(* Schneider Machine Expert - Basic project 13_counter_simulation, file version 3.0.0.0 *)
(* ProjectInformations: Name=New project *)

HARDWARE
  Cpu 0: TM221CE16R
  EthernetConfiguration: NetworkName=M221, IpAllocationMode=FixedAddress, IpAddress=0.0.0.0, SubnetMask=0.0.0.0
  SerialLineConfiguration: Baud=Baud19200, Parity=ParityEven, DataBits=DataBits8, StopBits=StopBits1, PhysicalMedium=PhysicalMediumRs485, TransmissionMode=TransmissionModeModbusRtu, SlaveId=1, Addressing=SlaveAddressing
  MastTask: UsePeriodScanMode=false, PeriodScan=100
  FastTask: Period=255
  CpuBehavior: StartingMode=StartAsPreviousState, AutoSaveRamOnEeprom=true, WatchdogPeriod=250

SYMBOLS  (address, symbol, comment, settings)
  %C0         [Preset=3]
  %C1         [Preset=3]
  %C2         [Preset=3]

POU New POU
  (* SectionNumber=1 *)

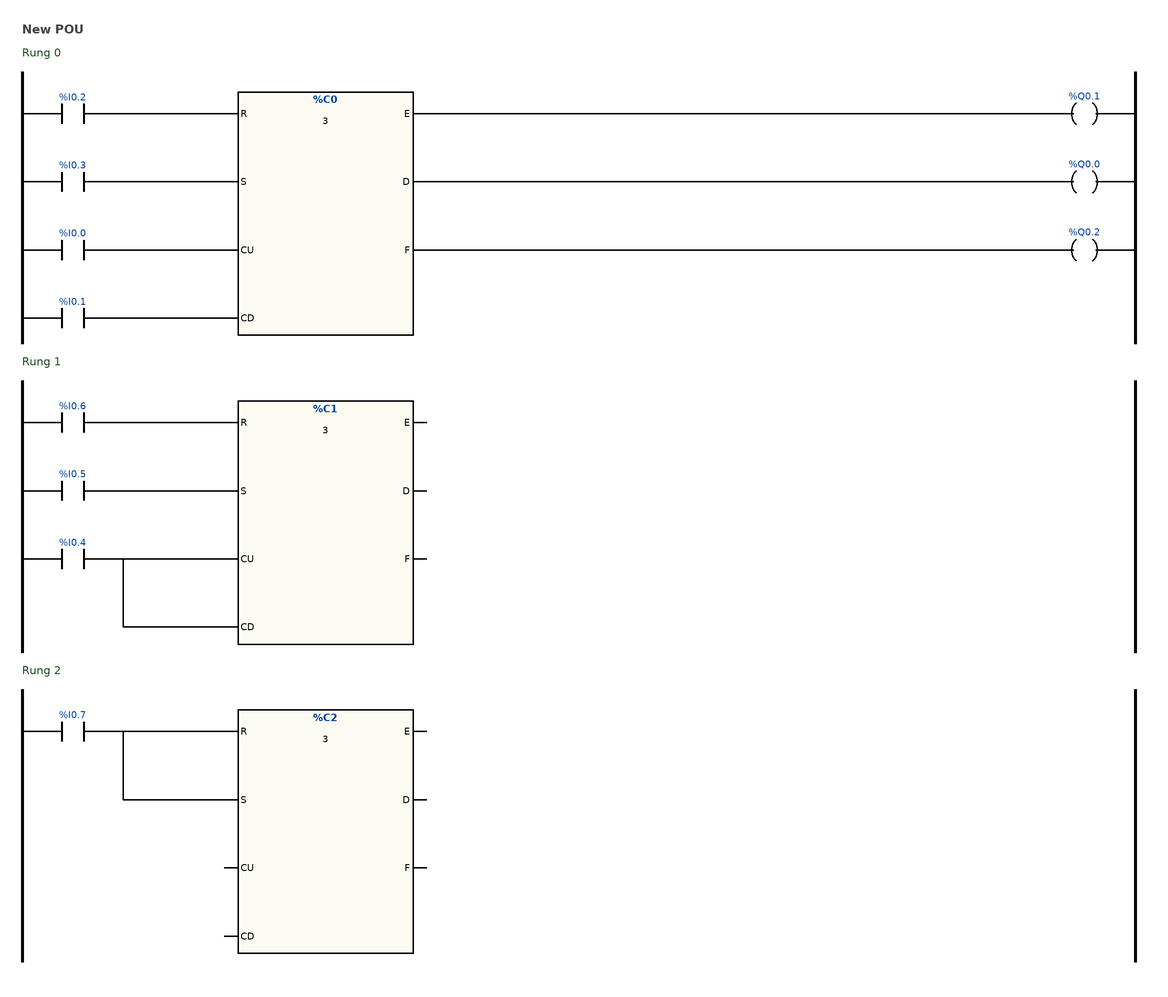

// Rung 0
  BLK %C0
  LD %I0.2
  R
  LD %I0.3
  S
  LD %I0.0
  CU
  LD %I0.1
  CD
  OUT_BLK
  LD E
  ST %Q0.1
  LD D
  ST %Q0.0
  LD F
  ST %Q0.2
  END_BLK
  // as ST:
  //   %C0(R := %I0.2, S := %I0.3, CU := %I0.0, CD := %I0.1);
  //   %Q0.1 := %C0.E;
  //   %Q0.0 := %C0.D;
  //   %Q0.2 := %C0.F;

// Rung 1
  BLK %C1
  LD %I0.6
  R
  LD %I0.5
  S
  LD %I0.4
  CU
  CD
  END_BLK
  // as ST:
  //   %C1(R := %I0.6, S := %I0.5, CU := %I0.4, CD := %I0.4);

// Rung 2
  BLK %C2
  LD %I0.7
  R
  S
  END_BLK
  // as ST:
  //   %C2(R := %I0.7, S := %I0.7);
